% RSLogix 500 project 3_pump_sequencing.RSS, saved by version 8.30.00.16 %
PROJECT "UNTITLED"    % processor: Bul.1763 MicroLogix 1100 Series A %

PROGRAM FILES
  LAD 2 "MAIN"  5 rungs
  LAD 215 "INPUT_MAP"  15 rungs  % Map data from discrete inputs to input map in N255 %
  LAD 225 "ONOFFSQTYP"  5 rungs  % Logic turning seq types lead, lag1, lag2 on or off %
  LAD 234 "LEADLAGLAG"  13 rungs  % Logic to assign sequence types to physical pumps %
  LAD 235 "ONOFFPUMPS"  5 rungs  % Logic for Pump 1/2/3 on-off assignments %
  LAD 244 "ONTMMINMAX"  6 rungs  % Calculate max and min ON times for pumps in Auto %
  LAD 245 "ONTM_ACCUM"  5 rungs  % Accumulate ON times, i.e. runtimes, for all pumps %
  LAD 255 "MANAUTOMNT"  6 rungs  % Which pumps are in Auto, Manual, or Maintenance? %

DATA FILES
  O0 OUTPUT  4 elements
  I1 INPUT  6 elements
  S2 STATUS  66 elements
  B3 BINARY  1 elements
  T4 TIMER  4 elements
  C5 COUNTER  1 elements
  R6 CONTROL  1 elements
  N7 INTEGER  1 elements
  F8 FLOAT  1 elements
  N200 MISC_INTS  1 elements
  B235 ONOFFLOGIC  1 elements
  L244 ONTMMINMAX  4 elements  % Maximum and minimum ON times for pumps in Auto %
  L245 ONTM_LONGS  6 elements  % Cumulative scan times and ON times for pumps %
  N254 BIT_COUNTS  8 elements  % Number of 1-bits for each INT value [0:7] %
  N255 MANAUTOMNT  14 elements  % Manual/Auto/Maintenance states of pumps %

LADDER 2 "MAIN"
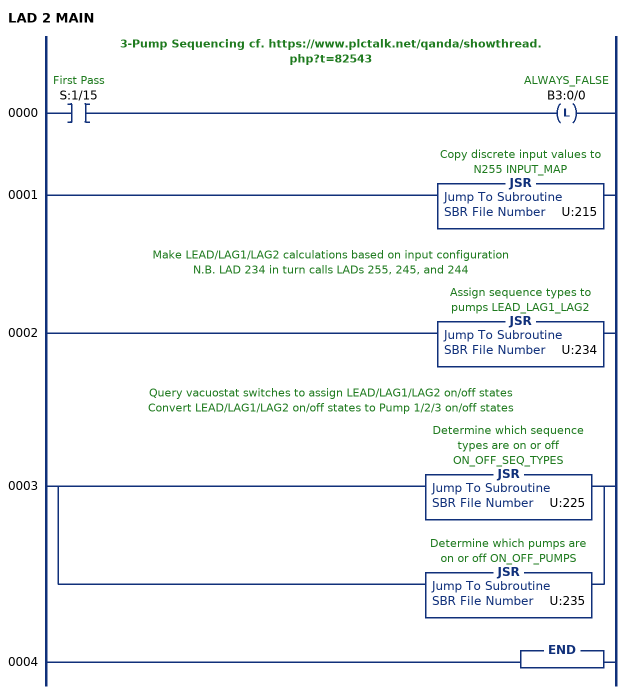
% Rung: 0 %
% TITLE: 3-Pump Sequencing cf. https://www.plctalk.net/qanda/showthread.php?t=82543 %
SOR XIC S:1/15 OTL B3:0/0 EOR
%   S:1/15  "First Pass" %
%   B3:0/0  ALWAYS_FALSE %
% Rung: 1 %
SOR JSR U:215 EOR
%   U:215  INPUT_MAP  "Copy discrete input values to N255" %
% Rung: 2 %
% Make LEAD/LAG1/LAG2 calculations based on input configuration
% N.B. LAD 234 in turn calls LADs 255, 245, and 244 %
SOR JSR U:234 EOR
%   U:234  LEAD_LAG1_LAG2  "Assign sequence types to pumps" %
% Rung: 3 %
% Query vacuostat switches to assign LEAD/LAG1/LAG2 on/off states
% Convert LEAD/LAG1/LAG2 on/off states to Pump 1/2/3 on/off states %
SOR BST JSR U:225 NXB JSR U:235 BND EOR
%   U:225  ON_OFF_SEQ_TYPES  "Determine which sequence types are on or off" %
%   U:235  ON_OFF_PUMPS  "Determine which pumps are on or off" %
% Rung: 4 %
SOR END EOR

LADDER 215 "INPUT_MAP"    % Map data from discrete inputs to input map in N255 %
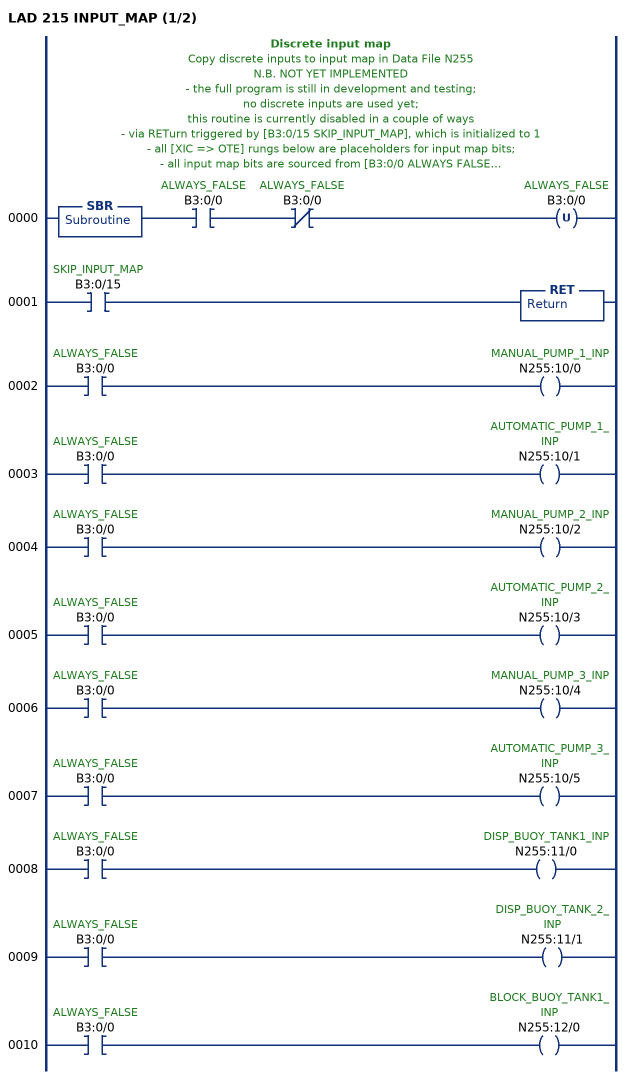
% Rung: 0 %
% TITLE: Discrete input map %
% Copy discrete inputs to input map in Data File N255
% 
% N.B. NOT YET IMPLEMENTED
% - the full program is still in development and testing;
% no discrete inputs are used yet;
% this routine is currently disabled in a couple of ways
%   - via RETurn triggered by [B3:0/15 SKIP_INPUT_MAP], which is initialized to 1
%   - all [XIC => OTE] rungs below are placeholders for input map bits;
%     - all input map bits are sourced from [B3:0/0 ALWAYS FALSE]
%       - so should the value of B3:0/15 become 1, all input map bits will be 0 %
SOR SBR XIC B3:0/0 XIO B3:0/0 OTU B3:0/0 EOR
%   B3:0/0  ALWAYS_FALSE %
% Rung: 1 %
SOR XIC B3:0/15 RET EOR
%   B3:0/15  SKIP_INPUT_MAP %
% Rung: 2 %
SOR XIC B3:0/0 OTE N255:10/0 EOR
%   B3:0/0  ALWAYS_FALSE %
%   N255:10/0  MANUAL_PUMP_1_INP %
% Rung: 3 %
SOR XIC B3:0/0 OTE N255:10/1 EOR
%   B3:0/0  ALWAYS_FALSE %
%   N255:10/1  AUTOMATIC_PUMP_1_INP %
% Rung: 4 %
SOR XIC B3:0/0 OTE N255:10/2 EOR
%   B3:0/0  ALWAYS_FALSE %
%   N255:10/2  MANUAL_PUMP_2_INP %
% Rung: 5 %
SOR XIC B3:0/0 OTE N255:10/3 EOR
%   B3:0/0  ALWAYS_FALSE %
%   N255:10/3  AUTOMATIC_PUMP_2_INP %
% Rung: 6 %
SOR XIC B3:0/0 OTE N255:10/4 EOR
%   B3:0/0  ALWAYS_FALSE %
%   N255:10/4  MANUAL_PUMP_3_INP %
% Rung: 7 %
SOR XIC B3:0/0 OTE N255:10/5 EOR
%   B3:0/0  ALWAYS_FALSE %
%   N255:10/5  AUTOMATIC_PUMP_3_INP %
% Rung: 8 %
SOR XIC B3:0/0 OTE N255:11/0 EOR
%   B3:0/0  ALWAYS_FALSE %
%   N255:11/0  DISP_BUOY_TANK1_INP %
% Rung: 9 %
SOR XIC B3:0/0 OTE N255:11/1 EOR
%   B3:0/0  ALWAYS_FALSE %
%   N255:11/1  DISP_BUOY_TANK_2_INP %
% Rung: 10 %
SOR XIC B3:0/0 OTE N255:12/0 EOR
%   B3:0/0  ALWAYS_FALSE %
%   N255:12/0  BLOCK_BUOY_TANK1_INP %

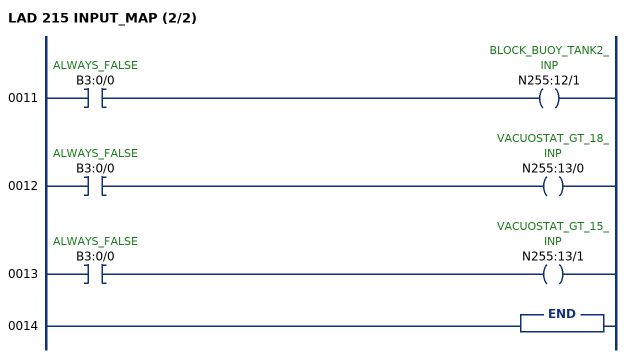
% Rung: 11 %
SOR XIC B3:0/0 OTE N255:12/1 EOR
%   B3:0/0  ALWAYS_FALSE %
%   N255:12/1  BLOCK_BUOY_TANK2_INP %
% Rung: 12 %
SOR XIC B3:0/0 OTE N255:13/0 EOR
%   B3:0/0  ALWAYS_FALSE %
%   N255:13/0  VACUOSTAT_GT_18_INP %
% Rung: 13 %
SOR XIC B3:0/0 OTE N255:13/1 EOR
%   B3:0/0  ALWAYS_FALSE %
%   N255:13/1  VACUOSTAT_GT_15_INP %
% Rung: 14 %
SOR END EOR

LADDER 225 "ONOFFSQTYP"    % Logic turning seq types lead, lag1, lag2 on or off %
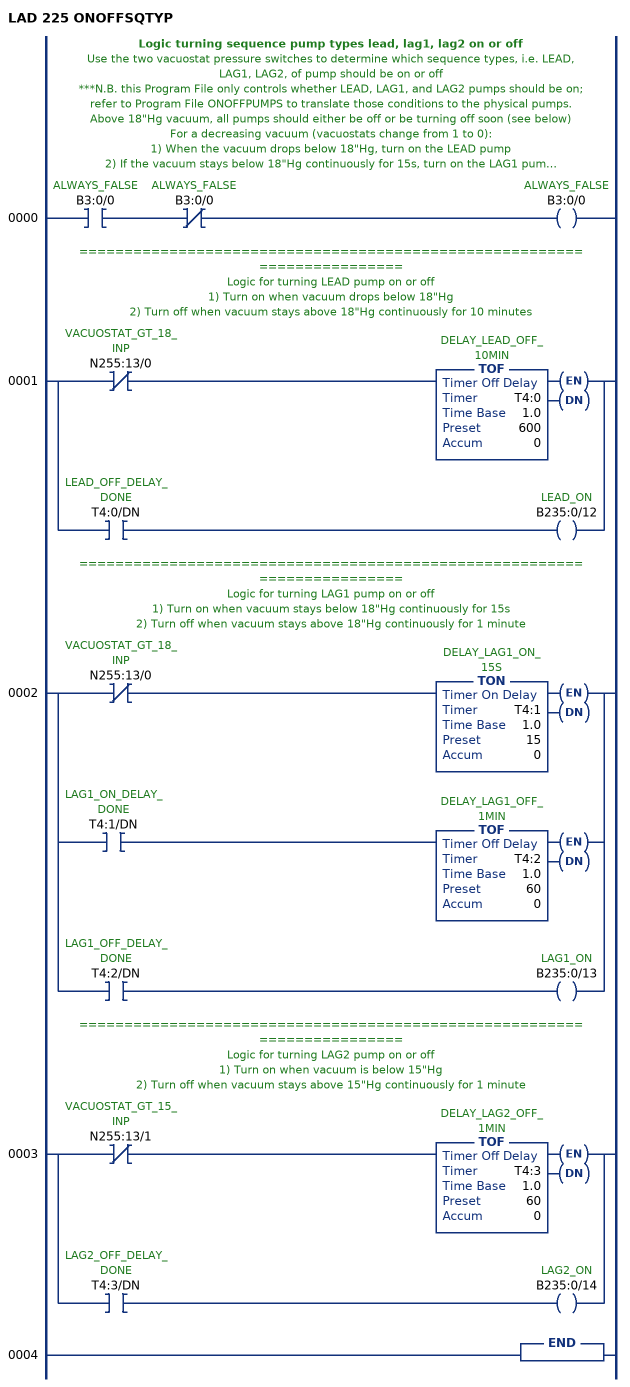
% Rung: 0 %
% TITLE: Logic turning sequence pump types lead, lag1, lag2 on or off %
% Use the two vacuostat pressure switches to determine which sequence types, i.e. LEAD, LAG1, LAG2, of pump should be on or off
% 
% ***N.B. this Program File only controls whether LEAD, LAG1, and LAG2 pumps should be on;
%            refer to Program File ONOFFPUMPS to translate those conditions to the physical pumps.
% 
% Above 18"Hg vacuum, all pumps should either be off or be turning off soon (see below)
% 
% For a decreasing vacuum (vacuostats change from 1 to 0):
% 1) When the vacuum drops below 18"Hg, turn on the LEAD pump
% 2) If the vacuum stays below 18"Hg continuously for 15s, turn on the LAG1 pump
% 3) If the vacuum drops below 15"Hg, turn on the LAG2 pump
% 
% For an increasing vacuum (vacuostats change from 0 to 1):
% 4) If vacuum stays above 15"Hg continuously for one minute, turn off the LAG2 pump,
% 5) If vacuum stays above 18"Hg continuously for fifteen seconds, turn off the LAG1 pump,
% 6) if vacuum stays above 18"Hg continuously for ten minutes, turn off the LEAD pump. %
SOR XIC B3:0/0 XIO B3:0/0 OTE B3:0/0 EOR
%   B3:0/0  ALWAYS_FALSE %
% Rung: 1 %
% ========================================================================
% Logic for turning LEAD pump on or off
% 1) Turn on when vacuum drops below 18"Hg
% 2) Turn off when vacuum stays above 18"Hg continuously for 10 minutes %
SOR BST XIO N255:13/0 TOF T4:0 1.0 600 0 NXB XIC T4:0/DN OTE B235:0/12 BND EOR
%   N255:13/0  VACUOSTAT_GT_18_INP %
%   T4:0  DELAY_LEAD_OFF_10MIN %
%   T4:0/DN  LEAD_OFF_DELAY_DONE %
%   B235:0/12  LEAD_ON %
% Rung: 2 %
% ========================================================================
% Logic for turning LAG1 pump on or off
% 1) Turn on when vacuum stays below 18"Hg continuously for 15s
% 2) Turn off when vacuum stays above 18"Hg continuously for 1 minute %
SOR BST XIO N255:13/0 TON T4:1 1.0 15 0 NXB XIC T4:1/DN TOF T4:2 1.0 60 0 NXB XIC T4:2/DN OTE B235:0/13 BND EOR
%   N255:13/0  VACUOSTAT_GT_18_INP %
%   T4:1  DELAY_LAG1_ON_15S %
%   T4:1/DN  LAG1_ON_DELAY_DONE %
%   T4:2  DELAY_LAG1_OFF_1MIN %
%   T4:2/DN  LAG1_OFF_DELAY_DONE %
%   B235:0/13  LAG1_ON %
% Rung: 3 %
% ========================================================================
% Logic for turning LAG2 pump on or off
% 1) Turn on when vacuum is below 15"Hg
% 2) Turn off when vacuum stays above 15"Hg continuously for 1 minute %
SOR BST XIO N255:13/1 TOF T4:3 1.0 60 0 NXB XIC T4:3/DN OTE B235:0/14 BND EOR
%   N255:13/1  VACUOSTAT_GT_15_INP %
%   T4:3  DELAY_LAG2_OFF_1MIN %
%   T4:3/DN  LAG2_OFF_DELAY_DONE %
%   B235:0/14  LAG2_ON %
% Rung: 4 %
SOR END EOR

LADDER 234 "LEADLAGLAG"    % Logic to assign sequence types to physical pumps %
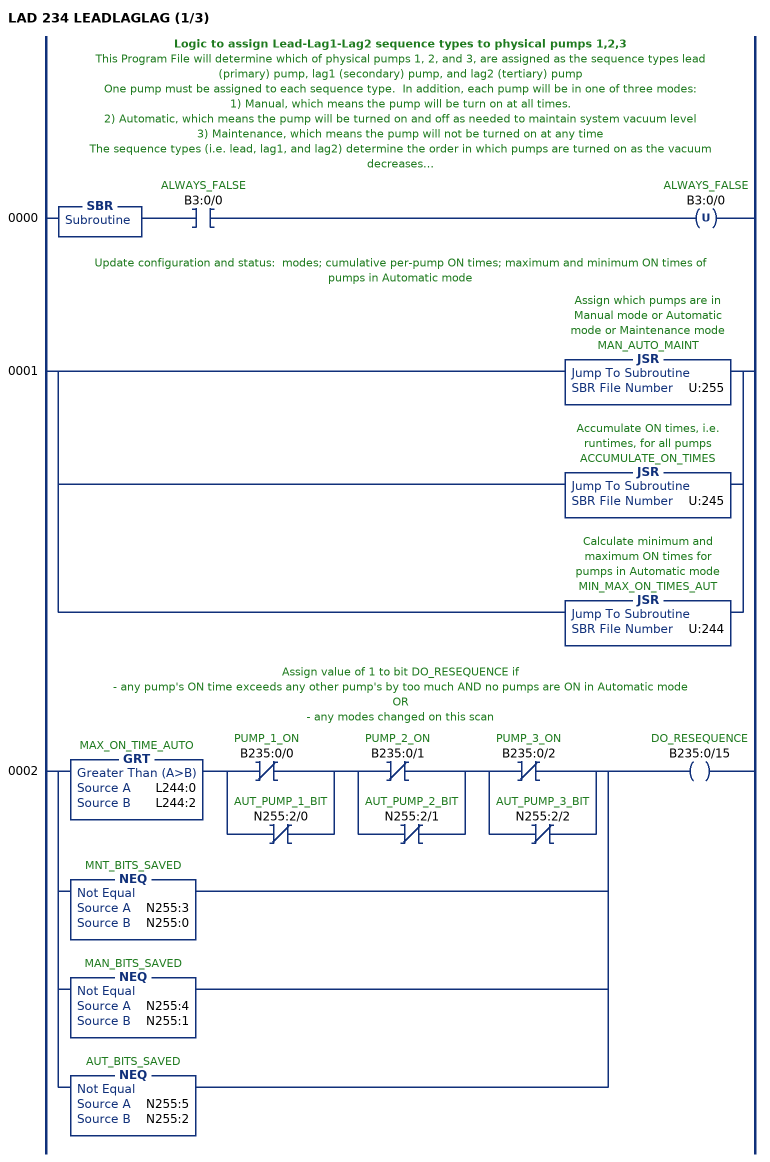
% Rung: 0 %
% TITLE: Logic to assign Lead-Lag1-Lag2 sequence types to physical pumps 1,2,3 %
% This Program File will determine which of physical pumps 1, 2, and 3, are assigned as the sequence types lead (primary) pump, lag1 (secondary) pump, and lag2 (tertiary) pump
% 
% One pump must be assigned to each sequence type.  In addition, each pump will be in one of three modes:
% 1) Manual, which means the pump will be turn on at all times.
% 2) Automatic, which means the pump will be turned on and off as needed to maintain system vacuum level
% 3) Maintenance, which means the pump will not be turned on at any time
% 
% The sequence types (i.e. lead, lag1, and lag2) determine the order in which pumps are turned on as the vacuum decreases.
% I.e. at first the lead pump will be turned on by itself, then lead+lag1 together, then lead+lag1+lag2 i.e. all together.
% 
% Merging this with the modes,
% - a pump in Manual mode is akin to the lead end of the sequence type progression (earlier on; later off)
% - a pump in Maintenance mode is akin to the lag2 end of the progression (later on; earlier off)
%   - Although a pump in Maintenance mode will never actually come on, it is still better to place it at the lag2 end so
%     pumps in all other modes will be turned on before the vacuum drops to the point that the lag2 pump is called to be on
% 
% With that in mind, the algorithm in this Program File will take the following approach:
% 
% Update pump modes, ON times, and maximum and minimum values of ON times for pumps in Automatic mode
% - if the lead/lag1/lag2 assignments are not to be changed on this scan (bit [RESEQUENCE] value is 0) , then keep all current assignments
% 
% If bit [RESEQUENCE] is 1, then fill in the following matrix with three 1s and six 0s:
% 
%               Pumps
%              1   2   3
%             ________
%   LEAD | A | B |  c |
%             -------------
%   LAG1  | g | h |  i  |
%              -------------
%   LAG2  | f  | E | D |
%              ------------
% 
% where
% - Each row will be assigned one 1 and two 0s, indicating one pump is assigned to that rows sequence type
% - Each column will be assigned one 1 and two 0s, indicating one sequence type is assigned to that column's pump
% - LEAD elements A and B are filled in first, favoring
%   - first the lowest-numbered pump in Manual mode if any exist,
%   - then the lowest-numbered pump in Automatic mode with the least ON time if any exist,
%   - finally pump 1 if all three pumps are in Maintenance mode
% - LAG2 elements D and E are filled in next, favoring
%   - first the highest-numbered pump in Maintenance mode if any exist,
%   - then the highest-numbered pump in Automatic mode with the most ON time if any exist
%   - finally pump3 if all three pumps are in Manual mode
% - All other elements c, f, g, h, i, will be filled in by difference, ensuring there is one 1-bit in each row and in each column %
SOR SBR XIC B3:0/0 OTU B3:0/0 EOR
%   B3:0/0  ALWAYS_FALSE %
% Rung: 1 %
% Update configuration and status:  modes; cumulative per-pump ON times; maximum and minimum ON times of pumps in Automatic mode %
SOR BST JSR U:255 NXB JSR U:245 NXB JSR U:244 BND EOR
%   U:255  MAN_AUTO_MAINT  "Assign which pumps are in Manual mode or Automatic mode or Maintenance mode" %
%   U:245  ACCUMULATE_ON_TIMES  "Accumulate ON times, i.e. runtimes, for all pumps" %
%   U:244  MIN_MAX_ON_TIMES_AUT  "Calculate minimum and maximum ON times for pumps in Automatic mode" %
% Rung: 2 %
% Assign value of 1 to bit DO_RESEQUENCE if
% - any pump's ON time exceeds any other pump's by too much AND no pumps are ON in Automatic mode
% OR
% - any modes changed on this scan %
SOR BST GRT L244:0 L244:2 BST XIO B235:0/0 NXB XIO N255:2/0 BND BST XIO B235:0/1 NXB XIO N255:2/1 BND BST XIO B235:0/2 NXB XIO N255:2/2 BND NXB NEQ N255:3 N255:0 NXB NEQ N255:4 N255:1 NXB NEQ N255:5 N255:2 BND OTE B235:0/15 EOR
%   L244:0  MAX_ON_TIME_AUTO %
%   L244:2  ONTIM_TO_RESEQUENCE %
%   B235:0/0  PUMP_1_ON %
%   N255:2/0  AUT_PUMP_1_BIT %
%   B235:0/1  PUMP_2_ON %
%   N255:2/1  AUT_PUMP_2_BIT %
%   B235:0/2  PUMP_3_ON %
%   N255:2/2  AUT_PUMP_3_BIT %
%   N255:3  MNT_BITS_SAVED %
%   N255:0  MNT_PUMP_BITS %
%   N255:4  MAN_BITS_SAVED %
%   N255:1  MAN_PUMP_BITS %
%   N255:5  AUT_BITS_SAVED %
%   N255:2  AUT_PUMP_BITS %
%   B235:0/15  DO_RESEQUENCE %

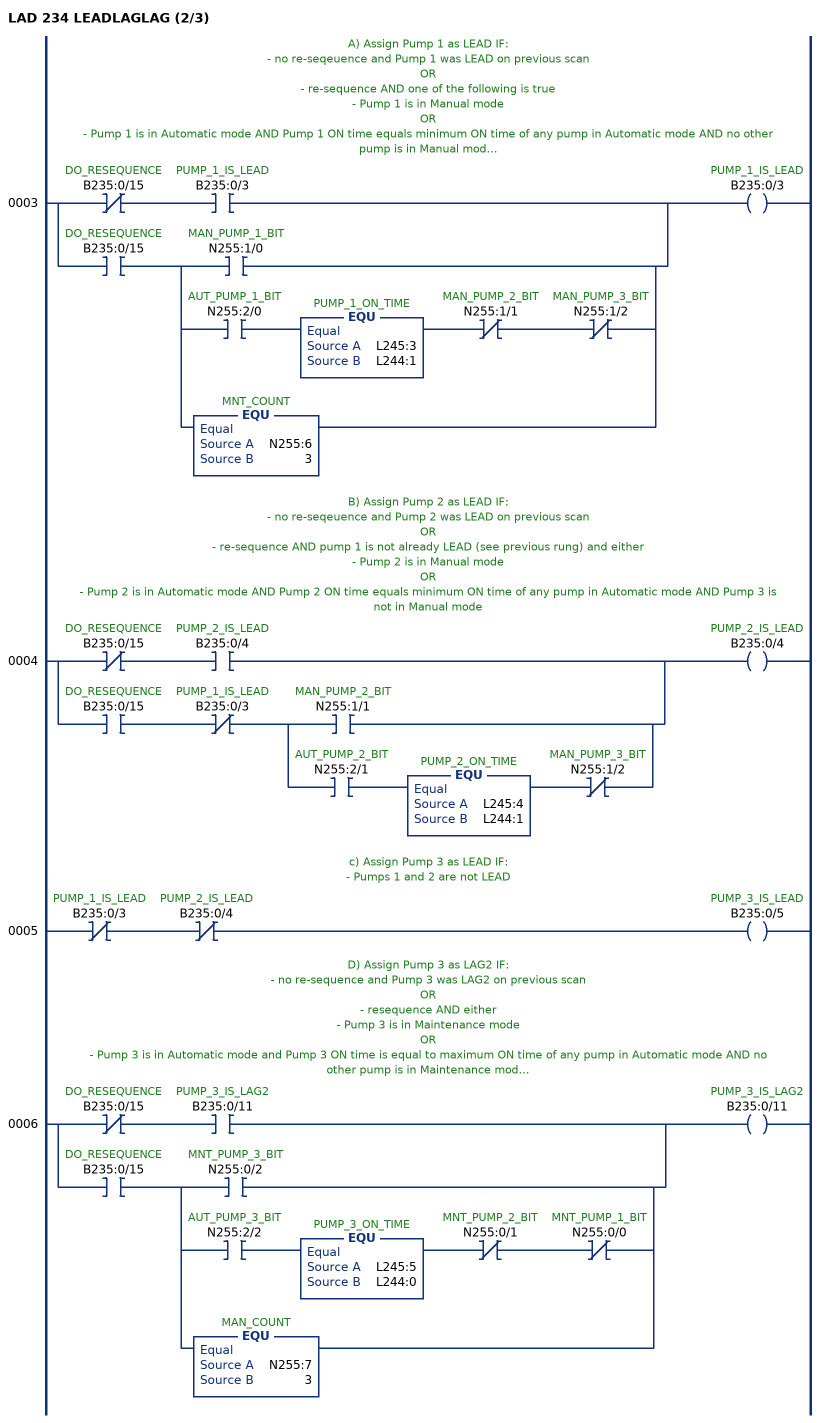
% Rung: 3 %
% A) Assign Pump 1 as LEAD IF:
% - no re-seqeuence and Pump 1 was LEAD on previous scan
% OR
% - re-sequence AND one of the following is true
%   - Pump 1 is in Manual mode
%   OR
%   - Pump 1 is in Automatic mode AND Pump 1 ON time equals minimum ON time of any pump in Automatic mode AND no other pump is in Manual mode
%   OR
%   - All 3 pumps are in maintenance mode %
SOR BST XIO B235:0/15 XIC B235:0/3 NXB XIC B235:0/15 BST XIC N255:1/0 NXB XIC N255:2/0 EQU L245:3 L244:1 XIO N255:1/1 XIO N255:1/2 NXB EQU N255:6 3 BND BND OTE B235:0/3 EOR
%   B235:0/15  DO_RESEQUENCE %
%   B235:0/3  PUMP_1_IS_LEAD %
%   N255:1/0  MAN_PUMP_1_BIT %
%   N255:2/0  AUT_PUMP_1_BIT %
%   L245:3  PUMP_1_ON_TIME %
%   L244:1  MIN_ON_TIME_AUTO %
%   N255:1/1  MAN_PUMP_2_BIT %
%   N255:1/2  MAN_PUMP_3_BIT %
%   N255:6  MNT_COUNT %
% Rung: 4 %
% B) Assign Pump 2 as LEAD IF:
% - no re-seqeuence and Pump 2 was LEAD on previous scan
% OR
% - re-sequence AND pump 1 is not already LEAD (see previous rung) and either
%   - Pump 2 is in Manual mode
%   OR
%   - Pump 2 is in Automatic mode AND Pump 2 ON time equals minimum ON time of any pump in Automatic mode AND Pump 3 is not in Manual mode %
SOR BST XIO B235:0/15 XIC B235:0/4 NXB XIC B235:0/15 XIO B235:0/3 BST XIC N255:1/1 NXB XIC N255:2/1 EQU L245:4 L244:1 XIO N255:1/2 BND BND OTE B235:0/4 EOR
%   B235:0/15  DO_RESEQUENCE %
%   B235:0/4  PUMP_2_IS_LEAD %
%   B235:0/3  PUMP_1_IS_LEAD %
%   N255:1/1  MAN_PUMP_2_BIT %
%   N255:2/1  AUT_PUMP_2_BIT %
%   L245:4  PUMP_2_ON_TIME %
%   L244:1  MIN_ON_TIME_AUTO %
%   N255:1/2  MAN_PUMP_3_BIT %
% Rung: 5 %
% c) Assign Pump 3 as LEAD IF:
% - Pumps 1 and 2 are not LEAD %
SOR XIO B235:0/3 XIO B235:0/4 OTE B235:0/5 EOR
%   B235:0/3  PUMP_1_IS_LEAD %
%   B235:0/4  PUMP_2_IS_LEAD %
%   B235:0/5  PUMP_3_IS_LEAD %
% Rung: 6 %
% D) Assign Pump 3 as LAG2 IF:
% - no re-sequence and Pump 3 was LAG2 on previous scan
% OR
% - resequence AND either
%   - Pump 3 is in Maintenance mode
%   OR
%   - Pump 3 is in Automatic mode and Pump 3 ON time is equal to maximum ON time of any pump in Automatic mode AND no other pump is in Maintenance mode
%   OR
%   - all pumps are in Manual mode %
SOR BST XIO B235:0/15 XIC B235:0/11 NXB XIC B235:0/15 BST XIC N255:0/2 NXB XIC N255:2/2 EQU L245:5 L244:0 XIO N255:0/1 XIO N255:0/0 NXB EQU N255:7 3 BND BND OTE B235:0/11 EOR
%   B235:0/15  DO_RESEQUENCE %
%   B235:0/11  PUMP_3_IS_LAG2 %
%   N255:0/2  MNT_PUMP_3_BIT %
%   N255:2/2  AUT_PUMP_3_BIT %
%   L245:5  PUMP_3_ON_TIME %
%   L244:0  MAX_ON_TIME_AUTO %
%   N255:0/1  MNT_PUMP_2_BIT %
%   N255:0/0  MNT_PUMP_1_BIT %
%   N255:7  MAN_COUNT %

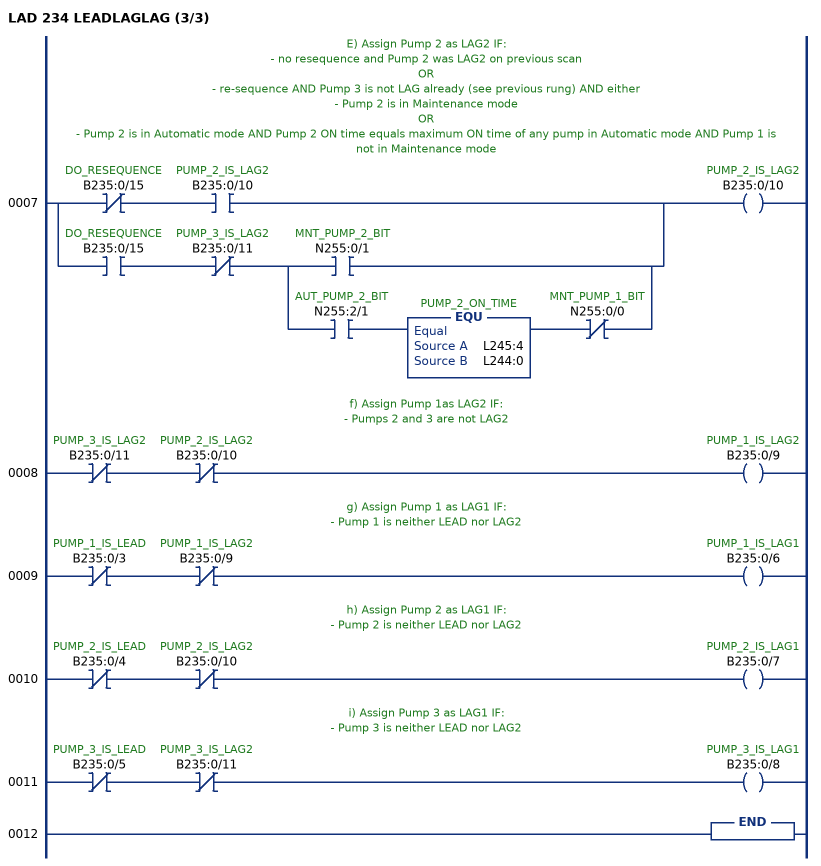
% Rung: 7 %
% E) Assign Pump 2 as LAG2 IF:
% - no resequence and Pump 2 was LAG2 on previous scan
% OR
% - re-sequence AND Pump 3 is not LAG already (see previous rung) AND either
%   - Pump 2 is in Maintenance mode
%   OR
%   - Pump 2 is in Automatic mode AND Pump 2 ON time equals maximum ON time of any pump in Automatic mode AND Pump 1 is not in Maintenance mode %
SOR BST XIO B235:0/15 XIC B235:0/10 NXB XIC B235:0/15 XIO B235:0/11 BST XIC N255:0/1 NXB XIC N255:2/1 EQU L245:4 L244:0 XIO N255:0/0 BND BND OTE B235:0/10 EOR
%   B235:0/15  DO_RESEQUENCE %
%   B235:0/10  PUMP_2_IS_LAG2 %
%   B235:0/11  PUMP_3_IS_LAG2 %
%   N255:0/1  MNT_PUMP_2_BIT %
%   N255:2/1  AUT_PUMP_2_BIT %
%   L245:4  PUMP_2_ON_TIME %
%   L244:0  MAX_ON_TIME_AUTO %
%   N255:0/0  MNT_PUMP_1_BIT %
% Rung: 8 %
% f) Assign Pump 1as LAG2 IF:
% - Pumps 2 and 3 are not LAG2 %
SOR XIO B235:0/11 XIO B235:0/10 OTE B235:0/9 EOR
%   B235:0/11  PUMP_3_IS_LAG2 %
%   B235:0/10  PUMP_2_IS_LAG2 %
%   B235:0/9  PUMP_1_IS_LAG2 %
% Rung: 9 %
% g) Assign Pump 1 as LAG1 IF:
% - Pump 1 is neither LEAD nor LAG2 %
SOR XIO B235:0/3 XIO B235:0/9 OTE B235:0/6 EOR
%   B235:0/3  PUMP_1_IS_LEAD %
%   B235:0/9  PUMP_1_IS_LAG2 %
%   B235:0/6  PUMP_1_IS_LAG1 %
% Rung: 10 %
% h) Assign Pump 2 as LAG1 IF:
% - Pump 2 is neither LEAD nor LAG2 %
SOR XIO B235:0/4 XIO B235:0/10 OTE B235:0/7 EOR
%   B235:0/4  PUMP_2_IS_LEAD %
%   B235:0/10  PUMP_2_IS_LAG2 %
%   B235:0/7  PUMP_2_IS_LAG1 %
% Rung: 11 %
% i) Assign Pump 3 as LAG1 IF:
% - Pump 3 is neither LEAD nor LAG2 %
SOR XIO B235:0/5 XIO B235:0/11 OTE B235:0/8 EOR
%   B235:0/5  PUMP_3_IS_LEAD %
%   B235:0/11  PUMP_3_IS_LAG2 %
%   B235:0/8  PUMP_3_IS_LAG1 %
% Rung: 12 %
SOR END EOR

LADDER 235 "ONOFFPUMPS"    % Logic for Pump 1/2/3 on-off assignments %
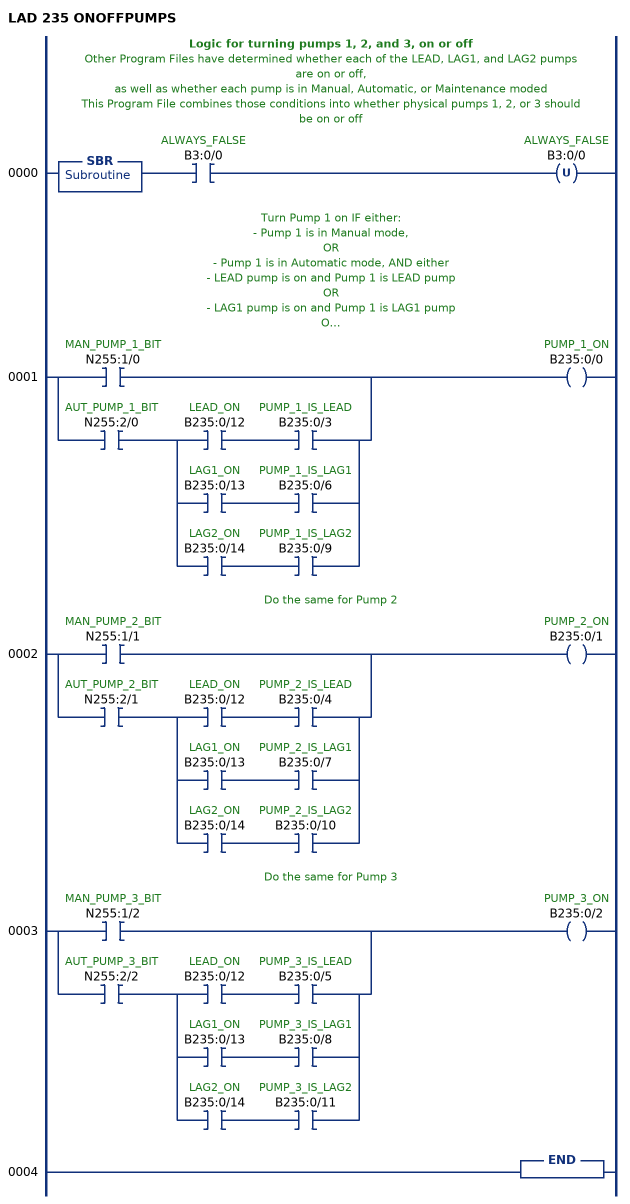
% Rung: 0 %
% TITLE: Logic for turning pumps 1, 2, and 3, on or off %
% Other Program Files have determined whether each of the LEAD, LAG1, and LAG2 pumps are on or off,
% as well as whether each pump is in Manual, Automatic, or Maintenance moded
% This Program File combines those conditions into whether physical pumps 1, 2, or 3 should be on or off %
SOR SBR XIC B3:0/0 OTU B3:0/0 EOR
%   B3:0/0  ALWAYS_FALSE %
% Rung: 1 %
% Turn Pump 1 on IF either:
% - Pump 1 is in Manual mode,
% OR
% - Pump 1 is in Automatic mode, AND either
%   - LEAD pump is on and Pump 1 is LEAD pump
%   OR
%   - LAG1 pump is on and Pump 1 is LAG1 pump
%   OR
%   - LAG2 pump is on and Pump 1 is LAG2 pump %
SOR BST XIC N255:1/0 NXB XIC N255:2/0 BST XIC B235:0/12 XIC B235:0/3 NXB XIC B235:0/13 XIC B235:0/6 NXB XIC B235:0/14 XIC B235:0/9 BND BND OTE B235:0/0 EOR
%   N255:1/0  MAN_PUMP_1_BIT %
%   N255:2/0  AUT_PUMP_1_BIT %
%   B235:0/12  LEAD_ON %
%   B235:0/3  PUMP_1_IS_LEAD %
%   B235:0/13  LAG1_ON %
%   B235:0/6  PUMP_1_IS_LAG1 %
%   B235:0/14  LAG2_ON %
%   B235:0/9  PUMP_1_IS_LAG2 %
%   B235:0/0  PUMP_1_ON %
% Rung: 2 %
% Do the same for Pump 2 %
SOR BST XIC N255:1/1 NXB XIC N255:2/1 BST XIC B235:0/12 XIC B235:0/4 NXB XIC B235:0/13 XIC B235:0/7 NXB XIC B235:0/14 XIC B235:0/10 BND BND OTE B235:0/1 EOR
%   N255:1/1  MAN_PUMP_2_BIT %
%   N255:2/1  AUT_PUMP_2_BIT %
%   B235:0/12  LEAD_ON %
%   B235:0/4  PUMP_2_IS_LEAD %
%   B235:0/13  LAG1_ON %
%   B235:0/7  PUMP_2_IS_LAG1 %
%   B235:0/14  LAG2_ON %
%   B235:0/10  PUMP_2_IS_LAG2 %
%   B235:0/1  PUMP_2_ON %
% Rung: 3 %
% Do the same for Pump 3 %
SOR BST XIC N255:1/2 NXB XIC N255:2/2 BST XIC B235:0/12 XIC B235:0/5 NXB XIC B235:0/13 XIC B235:0/8 NXB XIC B235:0/14 XIC B235:0/11 BND BND OTE B235:0/2 EOR
%   N255:1/2  MAN_PUMP_3_BIT %
%   N255:2/2  AUT_PUMP_3_BIT %
%   B235:0/12  LEAD_ON %
%   B235:0/5  PUMP_3_IS_LEAD %
%   B235:0/13  LAG1_ON %
%   B235:0/8  PUMP_3_IS_LAG1 %
%   B235:0/14  LAG2_ON %
%   B235:0/11  PUMP_3_IS_LAG2 %
%   B235:0/2  PUMP_3_ON %
% Rung: 4 %
SOR END EOR

LADDER 244 "ONTMMINMAX"    % Calculate max and min ON times for pumps in Auto %
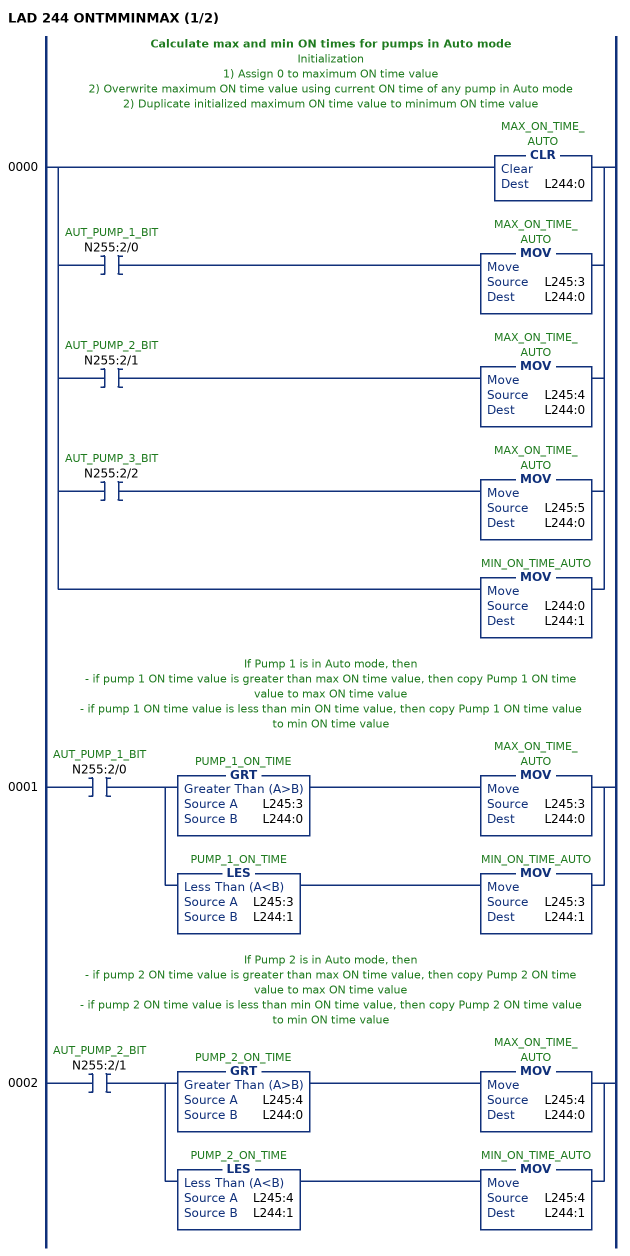
% Rung: 0 %
% TITLE: Calculate max and min ON times for pumps in Auto mode %
% Initialization
% 1) Assign 0 to maximum ON time value
% 2) Overwrite maximum ON time value using current ON time of any pump in Auto mode
% 2) Duplicate initialized maximum ON time value to minimum ON time value %
SOR BST CLR L244:0 NXB XIC N255:2/0 MOV L245:3 L244:0 NXB XIC N255:2/1 MOV L245:4 L244:0 NXB XIC N255:2/2 MOV L245:5 L244:0 NXB MOV L244:0 L244:1 BND EOR
%   L244:0  MAX_ON_TIME_AUTO %
%   N255:2/0  AUT_PUMP_1_BIT %
%   L245:3  PUMP_1_ON_TIME %
%   N255:2/1  AUT_PUMP_2_BIT %
%   L245:4  PUMP_2_ON_TIME %
%   N255:2/2  AUT_PUMP_3_BIT %
%   L245:5  PUMP_3_ON_TIME %
%   L244:1  MIN_ON_TIME_AUTO %
% Rung: 1 %
% If Pump 1 is in Auto mode, then
% - if pump 1 ON time value is greater than max ON time value, then copy Pump 1 ON time value to max ON time value
% - if pump 1 ON time value is less than min ON time value, then copy Pump 1 ON time value to min ON time value %
SOR XIC N255:2/0 BST GRT L245:3 L244:0 MOV L245:3 L244:0 NXB LES L245:3 L244:1 MOV L245:3 L244:1 BND EOR
%   N255:2/0  AUT_PUMP_1_BIT %
%   L245:3  PUMP_1_ON_TIME %
%   L244:0  MAX_ON_TIME_AUTO %
%   L244:1  MIN_ON_TIME_AUTO %
% Rung: 2 %
% If Pump 2 is in Auto mode, then
% - if pump 2 ON time value is greater than max ON time value, then copy Pump 2 ON time value to max ON time value
% - if pump 2 ON time value is less than min ON time value, then copy Pump 2 ON time value to min ON time value %
SOR XIC N255:2/1 BST GRT L245:4 L244:0 MOV L245:4 L244:0 NXB LES L245:4 L244:1 MOV L245:4 L244:1 BND EOR
%   N255:2/1  AUT_PUMP_2_BIT %
%   L245:4  PUMP_2_ON_TIME %
%   L244:0  MAX_ON_TIME_AUTO %
%   L244:1  MIN_ON_TIME_AUTO %

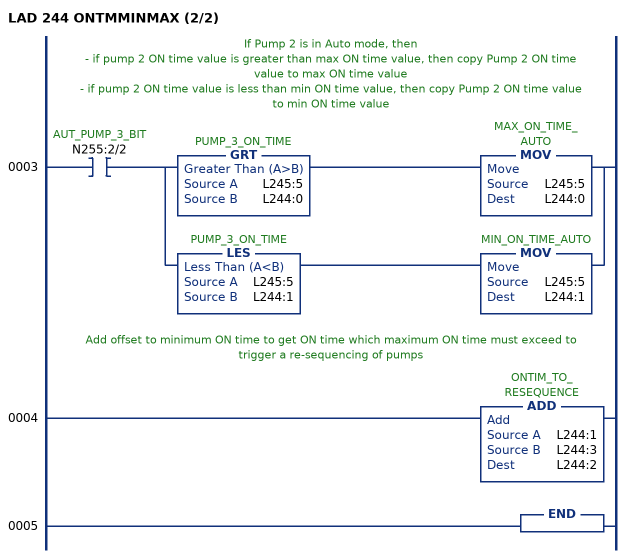
% Rung: 3 %
% If Pump 2 is in Auto mode, then
% - if pump 2 ON time value is greater than max ON time value, then copy Pump 2 ON time value to max ON time value
% - if pump 2 ON time value is less than min ON time value, then copy Pump 2 ON time value to min ON time value %
SOR XIC N255:2/2 BST GRT L245:5 L244:0 MOV L245:5 L244:0 NXB LES L245:5 L244:1 MOV L245:5 L244:1 BND EOR
%   N255:2/2  AUT_PUMP_3_BIT %
%   L245:5  PUMP_3_ON_TIME %
%   L244:0  MAX_ON_TIME_AUTO %
%   L244:1  MIN_ON_TIME_AUTO %
% Rung: 4 %
% Add offset to minimum ON time to get ON time which maximum ON time must exceed to trigger a re-sequencing of pumps %
SOR ADD L244:1 L244:3 L244:2 EOR
%   L244:1  MIN_ON_TIME_AUTO %
%   L244:3  ONTM_RESEQ_TRIGGER  "When Auto (max-min) on-time reaches this level, resequence" %
%   L244:2  ONTIM_TO_RESEQUENCE %
% Rung: 5 %
SOR END EOR

LADDER 245 "ONTM_ACCUM"    % Accumulate ON times, i.e. runtimes, for all pumps %
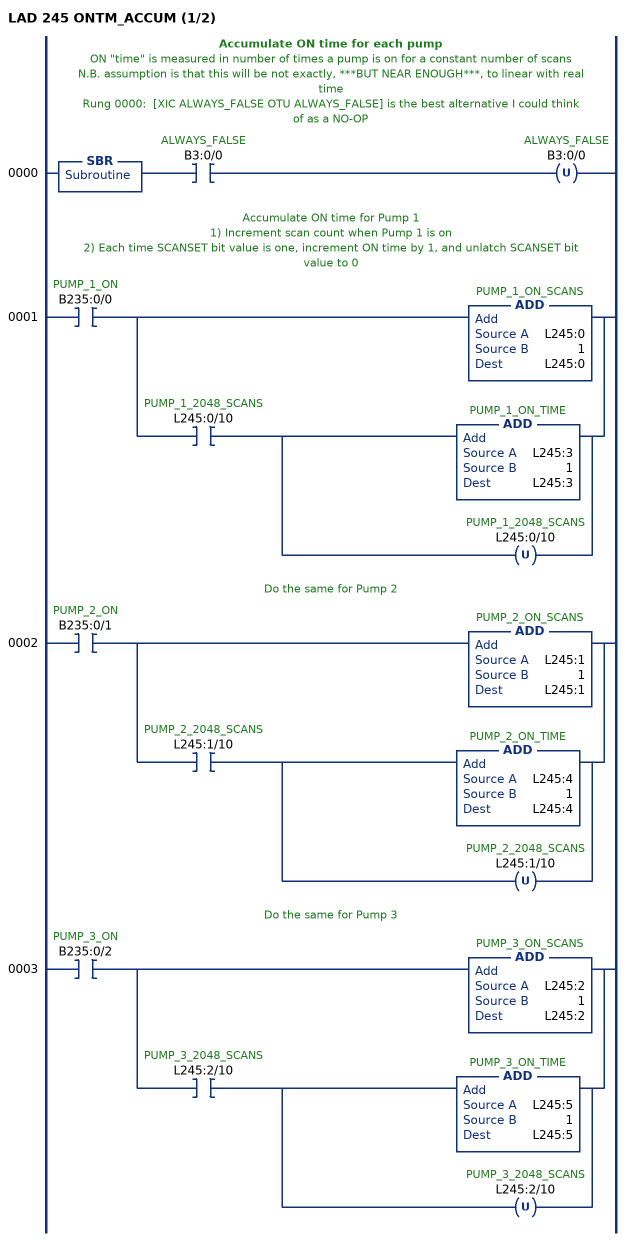
% Rung: 0 %
% TITLE: Accumulate ON time for each pump %
% ON "time" is measured in number of times a pump is on for a constant number of scans
% N.B. assumption is that this will be not exactly, ***BUT NEAR ENOUGH***, to linear with real time
% 
% Rung 0000:  [XIC ALWAYS_FALSE OTU ALWAYS_FALSE] is the best alternative I could think of as a NO-OP %
SOR SBR XIC B3:0/0 OTU B3:0/0 EOR
%   B3:0/0  ALWAYS_FALSE %
% Rung: 1 %
% Accumulate ON time for Pump 1
% 1) Increment scan count when Pump 1 is on
% 2) Each time SCANSET bit value is one, increment ON time by 1, and unlatch SCANSET bit value to 0 %
SOR XIC B235:0/0 BST ADD L245:0 1 L245:0 NXB XIC L245:0/10 BST ADD L245:3 1 L245:3 NXB OTU L245:0/10 BND BND EOR
%   B235:0/0  PUMP_1_ON %
%   L245:0  PUMP_1_ON_SCANS %
%   L245:0/10  PUMP_1_2048_SCANS %
%   L245:3  PUMP_1_ON_TIME %
% Rung: 2 %
% Do the same for Pump 2 %
SOR XIC B235:0/1 BST ADD L245:1 1 L245:1 NXB XIC L245:1/10 BST ADD L245:4 1 L245:4 NXB OTU L245:1/10 BND BND EOR
%   B235:0/1  PUMP_2_ON %
%   L245:1  PUMP_2_ON_SCANS %
%   L245:1/10  PUMP_2_2048_SCANS %
%   L245:4  PUMP_2_ON_TIME %
% Rung: 3 %
% Do the same for Pump 3 %
SOR XIC B235:0/2 BST ADD L245:2 1 L245:2 NXB XIC L245:2/10 BST ADD L245:5 1 L245:5 NXB OTU L245:2/10 BND BND EOR
%   B235:0/2  PUMP_3_ON %
%   L245:2  PUMP_3_ON_SCANS %
%   L245:2/10  PUMP_3_2048_SCANS %
%   L245:5  PUMP_3_ON_TIME %

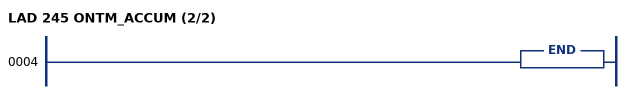
% Rung: 4 %
SOR END EOR

LADDER 255 "MANAUTOMNT"    % Which pumps are in Auto, Manual, or Maintenance? %
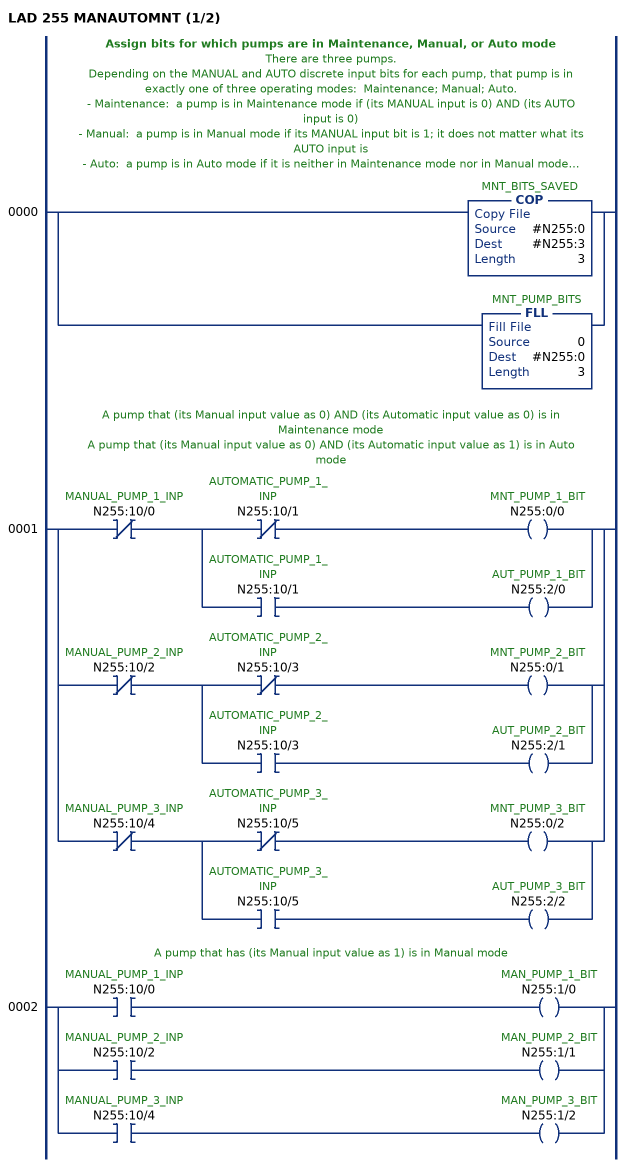
% Rung: 0 %
% TITLE: Assign bits for which pumps are in Maintenance, Manual, or Auto mode %
% There are three pumps.
% Depending on the MANUAL and AUTO discrete input bits for each pump, that pump is in exactly one of three operating modes:  Maintenance; Manual; Auto.
% - Maintenance:  a pump is in Maintenance mode if (its MANUAL input is 0) AND (its AUTO input is 0)
% - Manual:  a pump is in Manual mode if its MANUAL input bit is 1; it does not matter what its AUTO input is
% - Auto:  a pump is in Auto mode if it is neither in Maintenance mode nor in Manual mode; this is the same as if (its MANUAL input is 0) AND (its AUTO input is 1)
% 
% Initialization
% 1) COPy previous scans three sets of modes to saved modes
% 2) Clear what will become the current scan's three sets of modes %
SOR BST COP #N255:0 #N255:3 3 NXB FLL 0 #N255:0 3 BND EOR
%   N255:0  MNT_PUMP_BITS %
%   N255:3  MNT_BITS_SAVED %
% Rung: 1 %
% A pump that (its Manual input value as 0) AND (its Automatic input value as 0) is in Maintenance mode
% A pump that (its Manual input value as 0) AND (its Automatic input value as 1) is in Auto mode %
SOR BST XIO N255:10/0 BST XIO N255:10/1 OTE N255:0/0 NXB XIC N255:10/1 OTE N255:2/0 BND NXB XIO N255:10/2 BST XIO N255:10/3 OTE N255:0/1 NXB XIC N255:10/3 OTE N255:2/1 BND NXB XIO N255:10/4 BST XIO N255:10/5 OTE N255:0/2 NXB XIC N255:10/5 OTE N255:2/2 BND BND EOR
%   N255:10/0  MANUAL_PUMP_1_INP %
%   N255:10/1  AUTOMATIC_PUMP_1_INP %
%   N255:0/0  MNT_PUMP_1_BIT %
%   N255:2/0  AUT_PUMP_1_BIT %
%   N255:10/2  MANUAL_PUMP_2_INP %
%   N255:10/3  AUTOMATIC_PUMP_2_INP %
%   N255:0/1  MNT_PUMP_2_BIT %
%   N255:2/1  AUT_PUMP_2_BIT %
%   N255:10/4  MANUAL_PUMP_3_INP %
%   N255:10/5  AUTOMATIC_PUMP_3_INP %
%   N255:0/2  MNT_PUMP_3_BIT %
%   N255:2/2  AUT_PUMP_3_BIT %
% Rung: 2 %
% A pump that has (its Manual input value as 1) is in Manual mode %
SOR BST XIC N255:10/0 OTE N255:1/0 NXB XIC N255:10/2 OTE N255:1/1 NXB XIC N255:10/4 OTE N255:1/2 BND EOR
%   N255:10/0  MANUAL_PUMP_1_INP %
%   N255:1/0  MAN_PUMP_1_BIT %
%   N255:10/2  MANUAL_PUMP_2_INP %
%   N255:1/1  MAN_PUMP_2_BIT %
%   N255:10/4  MANUAL_PUMP_3_INP %
%   N255:1/2  MAN_PUMP_3_BIT %

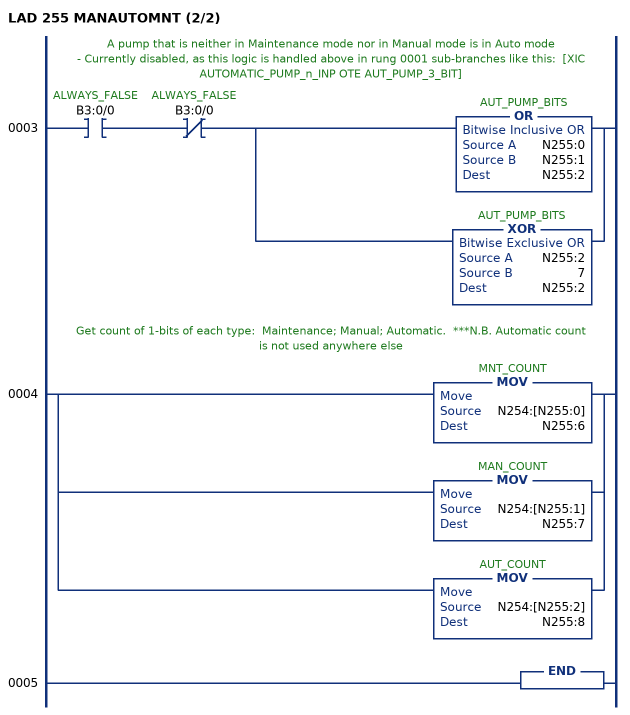
% Rung: 3 %
% A pump that is neither in Maintenance mode nor in Manual mode is in Auto mode
% - Currently disabled, as this logic is handled above in rung 0001 sub-branches like this:  [XIC AUTOMATIC_PUMP_n_INP OTE AUT_PUMP_3_BIT] %
SOR XIC B3:0/0 XIO B3:0/0 BST OR N255:0 N255:1 N255:2 NXB XOR N255:2 7 N255:2 BND EOR
%   B3:0/0  ALWAYS_FALSE %
%   N255:0  MNT_PUMP_BITS %
%   N255:1  MAN_PUMP_BITS %
%   N255:2  AUT_PUMP_BITS %
% Rung: 4 %
% Get count of 1-bits of each type:  Maintenance; Manual; Automatic.  ***N.B. Automatic count is not used anywhere else %
SOR BST MOV N254:[N255:0] N255:6 NXB MOV N254:[N255:1] N255:7 NXB MOV N254:[N255:2] N255:8 BND EOR
%   N255:0  MNT_PUMP_BITS %
%   N255:6  MNT_COUNT %
%   N255:1  MAN_PUMP_BITS %
%   N255:7  MAN_COUNT %
%   N255:2  AUT_PUMP_BITS %
%   N255:8  AUT_COUNT %
% Rung: 5 %
SOR END EOR

OTHER DOCUMENTED ADDRESSES
  N7:1  "Mask Result"
  N7:2  BITS_TO_SHIFT_RIGHT
  N7:3  DIVISOR
  N7:4  SHIFTED_SIGN_BIT_POS
  N254:0  "0=000b; zero 1-bits"
  N254:1  "1=001b; one 1-bit"
  N254:2  "2=010b; one 1-bit"
  N254:3  "3=011b; two 1-bits"
  N254:4  "4=100b; one 1-bit"
  N254:5  "5=101b; two 1-bits"
  N254:6  "6=110b; two 1-bits"
  N254:7  "7=111b; three 1-bits"
  N255:10  MNT_MAN_AUT_INPUTMAP
  N255:11  DISPOS_BUOY_INPUTMAP
  N255:12  BLOCK_BUOY_INPUTMAP
  N255:13  VACUOSTAT_INPUTMAP
  PFILE:244  "Calculate max & min ON times for pumps i n Auto"
  PFILE:254  "Runtime calculations for pumps in auto m ode"

COMMENTS NOT ATTACHED TO A CURRENT RUNG
  L245:7: Start calculation of MAX_ON_TIME_AUTO and MIN_ON_TIME_AUTO
    - these are maximum and minimum values of accumulated ON times any pumps that are in Auto mode
    
    Step 1) Initialize MAX_ON_TIME_AUTO and MIN_ON_TIME_AUTO to PUMP_n_ON_TIME of any pumps in Auto mode
                 or to 0 if no pumps are in Auto mode

DATA TABLE (non-zero values as saved)
DATA B3
% B3:0 % 0X8000
DATA T4
% .PRE .ACC %
% T4:0 % 600 0
% T4:1 % 15 0
% T4:2 % 60 0
% T4:3 % 60 0
DATA R6
% .LEN .POS %
% R6:0 % 128 0
DATA L244
% L244:0 % 0 0 0 300
DATA N254
% N254:0 % 0 1 1 2 1 2 2 3
